FUNCTION_BLOCK Process EXTENDS FB_PackML_BaseModule
VAR
	CurrentCustomMode : E_PMLCustomMode;
END_VAR

METHOD CyclicLogic
VAR
	_Start : BOOL;
END_VAR
IF NOT _InitComplete THEN
	_InitComplete := Initialize();
	RETURN;
END_IF

CurrentCustomMode := _CurrentMode;

//
SUPER^.CyclicLogic();
END_METHOD

END_FUNCTION_BLOCK

(* stored: Version 1.1.0.1
   POU Process: Id {83f7c65b-5908-4bc0-9481-015c3317f485}, SpecialFunc None
   Method CyclicLogic: Id {3b17b93b-5a6d-4d53-85b6-5a07dcaa6b32} *)
